(* CoDeSys 2.3 export: GetNextWritePointer.EXP *)

(* POU core/evt/GetNextWritePointer, ST *)
FUNCTION GetNextWritePointer : DINT
VAR_INPUT
    Length: DINT;
    WritePointer: DINT;
    ReadPointer: DINT;
    BufferSize: DINT;
END_VAR
VAR_IN_OUT
    BufferOverflow: DINT;
END_VAR
VAR
END_VAR
GetNextWritePointer := -1;
IF WritePointer >= ReadPointer THEN
    IF WritePointer + Length >= BufferSize THEN
        IF ReadPointer >= Length THEN
            BufferOverflow := WritePointer;
            GetNextWritePointer := 0;
        END_IF
    ELSE
        GetNextWritePointer := WritePointer + 1;
    END_IF
ELSIF ReadPointer - WritePointer > Length THEN
    GetNextWritePointer := WritePointer + 1;
END_IF
END_FUNCTION
